(* IEC 61131-3 sources: rust-plc/playground/multi_file_project/controllers, 2 files *)

(* ---- conveyor.st ---- *)
(*
 * Conveyor controller — manages belt movement.
 * Uses stdlib timers with TIME values.
 *)

FUNCTION_BLOCK ConveyorController
VAR_INPUT
    run_cmd : BOOL;
    speed_setpoint : INT;
END_VAR
VAR_OUTPUT
    motor_running : BOOL;
    current_speed : INT;
END_VAR
VAR
    ramp_timer : TON;
    ramp_step : INT := 0;
END_VAR
    IF run_cmd THEN
        motor_running := TRUE;
        // Ramp up speed gradually
        ramp_timer(IN1 := current_speed < speed_setpoint, PT := T#100ms);
        IF ramp_timer.Q THEN
            IF current_speed < speed_setpoint THEN
                current_speed := current_speed + 1;
            END_IF;
        END_IF;
    ELSE
        motor_running := FALSE;
        current_speed := 0;
    END_IF;
END_FUNCTION_BLOCK

(* ---- fill_controller.st ---- *)
(*
 * Fill controller — manages the bottle filling process.
 * Uses CTU from stdlib and types from types/process_data.st.
 *)

FUNCTION_BLOCK FillController
VAR_INPUT
    start : BOOL;
    target_fill : INT;
END_VAR
VAR_OUTPUT
    valve_open : BOOL;
    fill_done : BOOL;
    fill_count : INT;
END_VAR
VAR
    counter : CTU;
    filling : BOOL := FALSE;
    edge : R_TRIG;
    pulse_toggle : BOOL := FALSE;
END_VAR
    edge(CLK := start);

    IF edge.Q AND NOT filling THEN
        filling := TRUE;
        fill_count := 0;
        fill_done := FALSE;
    END_IF;

    pulse_toggle := NOT pulse_toggle;
    counter(CU := pulse_toggle AND filling, RESET := NOT filling, PV := target_fill);

    IF counter.Q THEN
        filling := FALSE;
        valve_open := FALSE;
        fill_done := TRUE;
    END_IF;

    fill_count := counter.CV;

    IF filling THEN
        valve_open := TRUE;
    ELSE
        valve_open := FALSE;
    END_IF;
END_FUNCTION_BLOCK
